RoboDK station: ProjetRobi (peinture de carrosserie de voiture).rdk

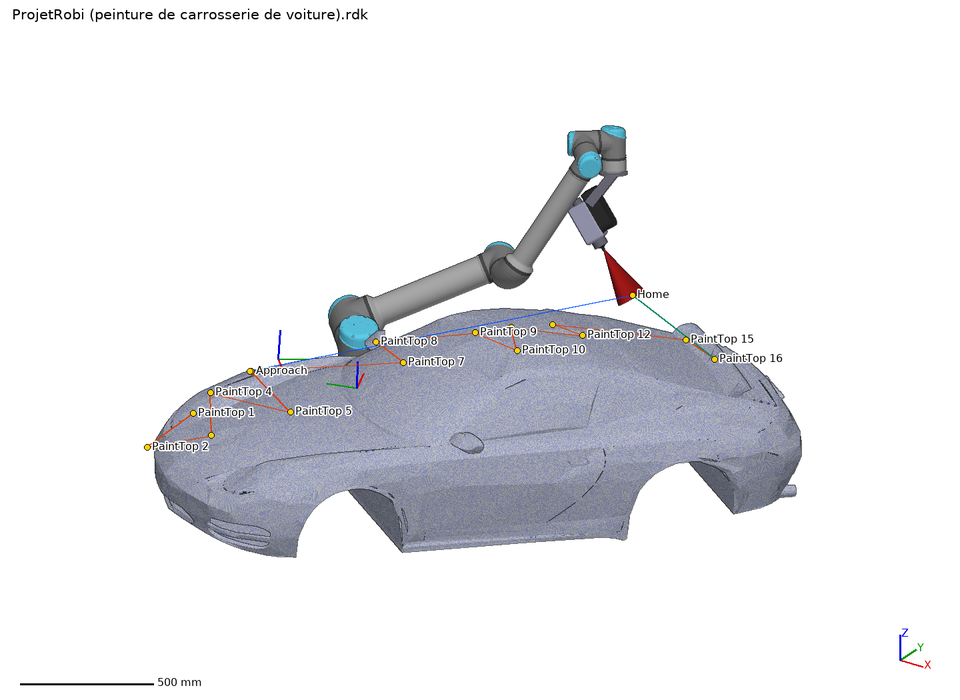
[picture v0: the station drawn from its stored meshes, robots at their saved joint values, targets as dots, program paths as lines]
Station ProjetRobi (saved by RoboDK 5.4.1). Poses are relative to the parent item; angles as X-Y-Z fixed-axis rotations.
  - frame UR10e Base at (-368.71, 170.53, 193.49) mm, rotated rx 2.68 ry -3.41 rz 111.7 deg
    - robot UR10e: 6 axes, payload 10 kg, reach 1300 mm, repeatability 0.05 mm, weight 28.9 kg
        modified DH rows (alpha deg, a mm, theta deg, d mm): 0, 0, 0, 180.7; 90, 0, 180, 0; 0, 612.6, 0, 0; 0, 571.335, 0, 174.15; -90, 0, 0, 119.85; 90, 0, 180, 116.55
        joint limits [-360, -360, -360, -360, -360, -360] to [360, 360, 360, 360, 360, 360]; home [0, -90, -90, 0, 90, 0]; saved at [113.16, -21.674, -38.197, 330.863, 252.01, 292.341]
      - tool Paint gun, TCP at (70, 0, 470) mm, rotated rx 0 ry 35 rz 0 deg, size 203.2 x 279.7 x 471.5 mm
  - frame Frame 2 at (-403.08, -291.14, 489.39) mm, rotated rx -4.04 ry -5.86 rz -48.03 deg
    - object Porsche911v0_123mm_IGS at (-1270, -3830, -960) mm, rotated rx 90.34 ry 4.9 rz 14.51 deg, size 1041.2 x 657.2 x 2494.3 mm, geometry from Porsche911v0_123mm_IGS.iges
    - target Home (Cartesian target) at (-312.59, 1365.82, 157.85) mm, rotated rx 171.28 ry -39.89 rz 76.1 deg; joints [86.717, -20.352, -51.977, 334.972, 253.509, 264.674] of UR10e
    - target Approach (Cartesian target) at (125.19, -117.62, -3.79) mm, rotated rx 173.29 ry -4.92 rz 71.06 deg; joints [-13.404, -78.768, 70.575, 254.775, 245.502, 165.829] of UR10e
    - target PaintTop 1 (Cartesian target) at (76.87, -319.1, -192.54) mm, rotated rx 100.06 ry -20.02 rz 121.55 deg; joints [-65.842, -52.915, 102.622, 193.293, 349.529, 126.048] of UR10e
    - target PaintTop 2 (Cartesian target) at (471.92, -541.76, -185.97) mm, rotated rx 152.11 ry 7.25 rz 156.75 deg; joints [-221.678, -125.303, -71.623, 321.784, 141.749, 74.568] of UR10e
    - target PaintTop 3 (Cartesian target) at (479.35, -302.79, -133.92) mm, rotated rx 164.57 ry -13.93 rz 174.37 deg; joints [-160.714, -112.475, -65.034, 300.368, 98.343, 102.628] of UR10e
    - target PaintTop 4 (Cartesian target) at (77.5, -258.54, -109.48) mm, rotated rx 124.07 ry 13.42 rz 135.72 deg; joints [-134.886, -205.679, -192.989, 209.539, 65.577, 148.941] of UR10e
    - target PaintTop 5 (Cartesian target) at (432.84, -3.48, -53.48) mm, rotated rx -179.78 ry -11.47 rz 135.62 deg; joints [-127.417, -163.41, -311.316, 217.631, 59.499, 164.671] of UR10e
    - target PaintTop 6 (Cartesian target) at (46.68, -110.04, -32.11) mm, rotated rx 163.14 ry 0.08 rz 132.07 deg; joints [-99.922, -169.373, -243.426, 149.622, 41.709, 201.203] of UR10e
    - target PaintTop 7 (Cartesian target) at (286.41, 430.28, 96.13) mm, rotated rx 170.01 ry -22.81 rz 135.99 deg; joints [51.715, -49.359, -347.573, 288.234, -107.371, 167.84] of UR10e
    - target PaintTop 8 (Cartesian target) at (-32.21, 369.22, 62.54) mm, rotated rx 156.8 ry 10.49 rz 121.35 deg; joints [108.795, -130.491, -241.973, 324.409, -138.317, 264.26] of UR10e
    - target PaintTop 9 (Cartesian target) at (244.48, 702.15, 203.07) mm, rotated rx 162.66 ry -4.2 rz 175.72 deg; joints [66.381, -51.454, -339.488, 262.274, -111.63, 137.353] of UR10e
    - target PaintTop 10 (Cartesian target) at (-288.98, 939.68, -57.32) mm, rotated rx 128.27 ry 43.82 rz 131.54 deg; joints [110.467, -12.772, -320.892, 207.555, -194.986, 176.275] of UR10e
    - target PaintTop 11 (Cartesian target) at (223.7, 837.61, 218.96) mm, rotated rx 179.17 ry -2.43 rz -135.85 deg; joints [72.393, -44.745, -354.195, 271.857, -101.738, 92.134] of UR10e
    - target PaintTop 12 (Cartesian target) at (-224.53, 1172.36, 28.33) mm, rotated rx -172.84 ry 14.11 rz -133.8 deg; joints [104.859, -39.695, -319.368, 226.879, -131.336, 106.964] of UR10e
    - target PaintTop 13 (Cartesian target) at (155.66, 1002.3, 208.38) mm, rotated rx -175.38 ry -4.92 rz -135.35 deg; joints [78.594, -44.151, -353.731, 275.034, -109.309, 94.553] of UR10e
    - target PaintTop 14 (Cartesian target) at (155.66, 1002.3, 208.38) mm, rotated rx -175.38 ry -4.92 rz -135.35 deg; joints [78.594, -44.151, -353.731, 275.034, -109.309, 94.553] of UR10e
    - target PaintTop 15 (Cartesian target) at (-140.11, 1552.32, 47) mm, rotated rx 153.8 ry 5.34 rz -140.39 deg; joints [90.542, -34.836, -335.135, 231.293, -98.146, 120.211] of UR10e
    - target PaintTop 16 (Cartesian target) at (62.15, 1636.34, 44.8) mm, rotated rx 138.86 ry -0.11 rz -135.62 deg; joints [78.378, -62.677, -286.081, 210.346, -74.181, 120.04] of UR10e
    - target Retract (Cartesian target) at (62.15, 1636.34, 44.8) mm, rotated rx 138.86 ry -0.11 rz -135.62 deg; joints [78.378, -62.677, 73.919, 210.346, 285.819, 120.04] of UR10e
  - Python program SprayOn (listed below)
  - program ApproachMove (4 instructions, listed below)
  - program Prog3 (18 instructions, listed below)
  - program Retract (4 instructions, listed below)
  - program MainProg (5 instructions, listed below)
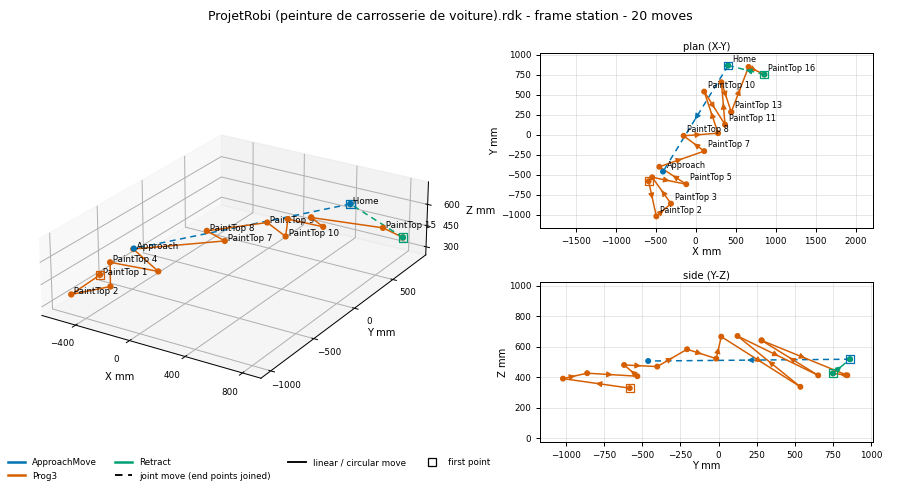
[picture p0: tool path of ProjetRobi (peinture de carrosserie de voiture).rdk in frame station, 20 of 20 moves have a stored position in this frame; points joined in program order, loops and branches not executed]

--- Python program SprayOn ---
# This macro allows simulating a spray gun for painting or to simulate the trace of inspaction
#
# You can call SprayOn(1) to simulate turning the Spray gun ON or SprayOn(0) to stop simulating the gun
# Calling SprayOn(-1) clears all displayed data
# The macro will output spray gun statistics
#
# --------------------------------------------------------------
# This script shows how to create "spray" object in RoboDK that allows simulating particle deposition by using:
# RDK.Spray_Add(tool, object, options_command, volume, geometry)
#    tool: tool item (TCP) to use
#    object: object to project the particles
#    options_command (optional): string to specify options.
#    volume (optional): Matrix of parameters defining the volume of the spray gun
#    geometry (optional): Matrix of vertices defining the triangles.
#
# More information here:
# https://robodk.com/doc/en/PythonAPI/robolink.html#robolink.Robolink.Spray_Add
# https://robodk.com/doc/en/RoboDK-API.html
#
# The scripts ArcStart, ArcEnd and WeldOn and SpindleOn behave in a similar way, the only difference is the default behavior
# This behavior simmulates Fanuc Arc Welding and triggers appropriate output when using the customized post processor.
# Select ESC to clear the trace manually.
#
# Example scripts that use Spray_Add:
#     SpindleOn / SpindleOff    -> Turn trace On/Off
#     ArcOn / ArcOff            -> Turn trace On/Off
#     SprayOn / SprayOff        -> Simulate a spray given a workspace volume (for painting)
#     WeldOn / WeldOff          -> Support for multiple weld guns

#------------------------------------------------------------------

# Use a specific tool as a spray gun
Tool_Name = None
#Tool_Name = 'Tool 2'

# Use a specific object to project particles:
Object_Name = None
#Object_Name = 'Part'



# Define the default action (0 to deactivate, +1 to activate, -1 to clear any spray gun simulation)
# Setting it to None will display a message
ACTION = None

from robolink import *    # API to communicate with RoboDK
from robodk import *      # basic matrix operations
RDK = Robolink()

# quit if we are not in simulation mode
if RDK.RunMode() != RUNMODE_SIMULATE:
    quit()

# Get any previously added spray gun simulations and display statistics (spray on the part vs spray falling out of the part)
info, data = RDK.Spray_GetStats()
if data.size(1) > 0:
    print("Spray gun statistics:")
    print(info)
    print(data.tr())
    # # Diplay statistics
    # RDK.ShowMessage("Material used: %.1f%%<br>Material waisted: %.1f%%<br>Total particles: %.1f" % (data[1,0],data[2,0],data[3,0]), True)
    # # Clear previous spray
    # RDK.Spray_Clear()

# Check if we are running this program inside another program and passing arguments
import sys
if len(sys.argv) > 1:
    ACTION = int(sys.argv[1])

# If the default ACTION is None, display a message to activate/deactivate the spray gun
if ACTION is None:
    print('Note: This macro can be called as Spray(1) or SprayOn(0)')
    entry = mbox('Turn gun ON or OFF', ('On', '1'), ('Off', '0'))
    if not entry:
        quit()
    ACTION = int(entry)

if ACTION == 0:
    # Turn the gun off
    RDK.Spray_SetState(SPRAY_OFF)

elif ACTION < 0:
    # Clear all spray simulations (same as pressing ESC key)
    RDK.Spray_Clear()

elif ACTION > 0:
    # Create a new spray gun object in RoboDK
    # by using RDK.Spray_Add(tool, object, options_command, volume, geometry)
    # tool: tool item (TCP) to use
    # object: object to project the particles
    # options_command (optional): string to specify options. Example:
    #     STEP=AxB: Defines the grid to be projected 1x1 means only one line of particle projection (for example, for welding)
    #     PARTICLE: Defines the shape and size of particle (sphere or particle), unless a specific geometry is provided:
    #       a- SPHERE(radius, facets)
    #       b- SPHERE(radius, facets, scalex, scaley, scalez)
    #       b- CUBE(sizex, sizey, sizez)
    #     RAND=factor: Defines a random factor factor 0 means that the particles are not deposited randomly
    #     ELLYPSE: defines the volume as an ellypse (default)
    #     RECTANGLE: defines the volume as a rectangle
    #     PROJECT: project the particles to the surface (default) (for welding, painting or scanning)
    #     NO_PROJECT: does not project the particles to the surface (for example, for 3D printing)
    #
    # volume (optional): Matrix of parameters defining the volume of the spray gun
    # geometry (optional): Matrix of vertices defining the triangles.


    tool = 0    # auto detect active tool
    obj = 0     # auto detect object in active reference frame
    if Tool_Name is not None:
        tool = RDK.Item(Tool_Name, ITEM_TYPE_TOOL)

    if Object_Name is not None:
        obj = RDK.Item(Object_Name, ITEM_TYPE_OBJECT)
    # We can specify a given tool object and/or object
    #robot = RDK.Item("ABB IRB 2600-12/1.85", ITEM_TYPE_ROBOT)
    #tools = robot.Childs()
    #if len(tools) > 0:
    #    tool = tools[0]
    #obj = RDK.Item('object', ITEM_TYPE_OBJECT)

    options_command = "ELLYPSE PROJECT PARTICLE=SPHERE(4,8,1,1,0.5) STEP=8x8 RAND=2" # simulate
    #options_command = "PARTICLE=CUBE(10,10,2) STEP=8x8"
    #options_command = "PARTICLE=SPHERE(4,8) STEP=8x8"
    #options_command = "PARTICLE=SPHERE(4,8,1,1,0.1) STEP=8x8 RAND=3"

    # Example commands for welding:
    # options_command = "PROJECT PARTICLE=SPHERE(4,8)"
    # options_command = PARTICLE=SPHERE(4,8) STEP=1x0


    # define the ellypse volume as p0, pA, pB, colorRGBA (close and far), in mm
    # coordinates must be provided with respect to the TCP
    close_p0 = [   0,   0, -200] # xyz in mm: Center of the conical ellypse (side 1)
    close_pA = [   5,   0, -200] # xyz in mm: First vertex of the conical ellypse (side 1)
    close_pB = [   0,  10, -200] # xyz in mm: Second vertex of the conical ellypse (side 1)
    close_color = [ 1, 0, 0, 1]  # RGBA (0-1)

    far_p0   = [   0,   0,  50] # xyz in mm: Center of the conical ellypse (side 2)
    far_pA   = [  60,   0,  50] # xyz in mm: First vertex of the conical ellypse (side 2)
    far_pB   = [   0, 120,  50] # xyz in mm: Second vertex of the conical ellypse (side 2)
    far_color   = [ 0, 0, 1, 0.2]  # RGBA (0-1)

    close_param = close_p0 + close_pA + close_pB + close_color
    far_param = far_p0 + far_pA + far_pB + far_color
    volume = Mat([close_param, far_param]).tr()
    RDK.Spray_Add(tool, obj, options_command, volume)
    RDK.Spray_SetState(SPRAY_ON)


    # Another example with a varying rectancular shape
    # define the rectangular volume as p0, pA, pB, colorRGBA (close and far)
    # close_param = [-90,-117,  0,  90,-117,0,   -90,117,  0,       0.2,0.2,1,.1]
    # far_param   = [-175,-190,200, 175,-190,200,   -175,190,200,   0.5,0,0,.9]
    # volume = Mat([close_param, far_param])
    # RDK.Spray_Add(tool, obj, "RECTANGLE PARTICLE=SPHERE(2,5) STEP=15x15 RAND=3", volume.tr())
    # RDK.Spray_SetState(SPRAY_ON)

    # Optional: define geometry as a list of triangles with normals (instead of a scaled cube or a sphere)
    # geom = Mat([[0,0,0,   0,0,1], [5,0,0,   0,0,1], [0,5,0,   0,0,1]])
    # RDK.Spray_Add(tool, obj, "STEP=8x8 RANDX=3", volume.tr(), geom.tr())
    # RDK.Spray_SetState(SPRAY_ON)

--- program ApproachMove (robot UR10e) ---
  Définir Ref.: Frame 2
  Choisir Outil: Paint gun
  MoveJ (Home)
  MoveJ (Approach)

--- program Prog3 (robot UR10e) ---
  Définir Ref.: Frame 2
  Choisir Outil: Paint gun
  MoveJ (PaintTop 1)
  MoveL (PaintTop 2)
  MoveL (PaintTop 3)
  MoveL (PaintTop 4)
  MoveL (PaintTop 5)
  MoveL (PaintTop 6)
  MoveL (PaintTop 7)
  MoveL (PaintTop 8)
  MoveL (PaintTop 9)
  MoveL (PaintTop 10)
  MoveL (PaintTop 11)
  MoveL (PaintTop 12)
  MoveL (PaintTop 13)
  MoveL (PaintTop 14)
  MoveL (PaintTop 15)
  MoveL (PaintTop 16)

--- program Retract (robot UR10e) ---
  Définir Ref.: Frame 2
  Choisir Outil: Paint gun
  MoveL (Retract)
  MoveJ (Home)

--- program MainProg (robot UR10e) ---
  Appel ApproachMove
  Appel SprayOn
  Appel Prog3
  Appel SprayOn
  Appel Retract
